// TwinCAT 3 PLC project Test
// ProgramVersion: 3.1.4023.0
// libraries:
//   Tc2_EtherCAT, * (Beckhoff Automation GmbH)
//   Tc2_SerialCom, * (Beckhoff Automation GmbH)
//   Tc2_Standard, * (Beckhoff Automation GmbH)
//   Tc2_System, * (Beckhoff Automation GmbH)
//   Tc2_Utilities, * (Beckhoff Automation GmbH)
//   Tc3_EventLogger, * (Beckhoff Automation GmbH)
//   Tc3_JsonXml, * (Beckhoff Automation GmbH)
//   Tc3_Module, * (Beckhoff Automation GmbH)
// project tree:
//   GVLs/ OperationControlData.TcGVL, Test.TcGVL, XMCData.TcGVL (not stored)
//   OOPs/ FB_HighLevelSystem.TcPOU (not stored), ITF_HighLevelSystem.TcIO (not stored), ITF_SubSystem.TcIO
//   / PlcTask.TcTTO
//   POUs/ MAIN.TcPOU
// real-time tasks:
//   TASK PlcTask: cycle T#1ms, priority 20, ADS port 350
// I/O:
//   DEVICE Gerät 4 (EtherCAT Slave), AmsNetId 10.183.66.136.5.255
// variable links:
//   Test/Test Instance <-> Device 4 (EtherCAT Slave)
//     PlcTask Outputs/Test.nTest <-> Outputs/Test

CONFIGURATION Test
    RESOURCE PLC ON TwinCAT3
        TASK PlcTask(INTERVAL := T#1ms, PRIORITY := 20);
        PROGRAM MAIN WITH PlcTask : MAIN;
    END_RESOURCE
END_CONFIGURATION

// ---- GVLs/OperationControlData.TcGVL
{attribute 'qualified_only'}
VAR_GLOBAL
	stFromOCToMC 			AT %I* : FromOperationControlToMainControl;
	
	stFromMCToOC 			AT %Q* : FromMainControlToOperationControl;
	stForwardXMC1ToOC 		AT %Q* : ForwardXMC1ToOperationControl;
	stForwardXMC2ToOC 		AT %Q* : ForwardXMC2ToOperationControl;
	stForwardXMC3ToOC 		AT %Q* : ForwardXMC3ToOperationControl;
	stForwardXMC4ToOC 		AT %Q* : ForwardXMC4ToOperationControl;
END_VAR

// ---- GVLs/Test.TcGVL
{attribute 'qualified_only'}
VAR_GLOBAL
	nTest AT %Q* : INT;
END_VAR

// ---- OOPs/ITF_SubSystem.TcIO
INTERFACE ITF_SubSystem

PROPERTY PUBLIC eCondition : SubLevelCondition
GET
END_GET
END_PROPERTY

PROPERTY PUBLIC nErrorID : UDINT
GET
END_GET
END_PROPERTY

END_INTERFACE

// ---- POUs/MAIN.TcPOU
PROGRAM MAIN
VAR
	fbTimer : TON;
	i : INT;
END_VAR

fbTimer(IN:=TRUE, PT:=T#5S);
IF fbTimer.Q THEN
	i := i + 1;
	fbTimer(IN := FALSE);
END_IF

Test.nTest := i;

END_PROGRAM
